RoboDK station: Colour sorting robot.rdk

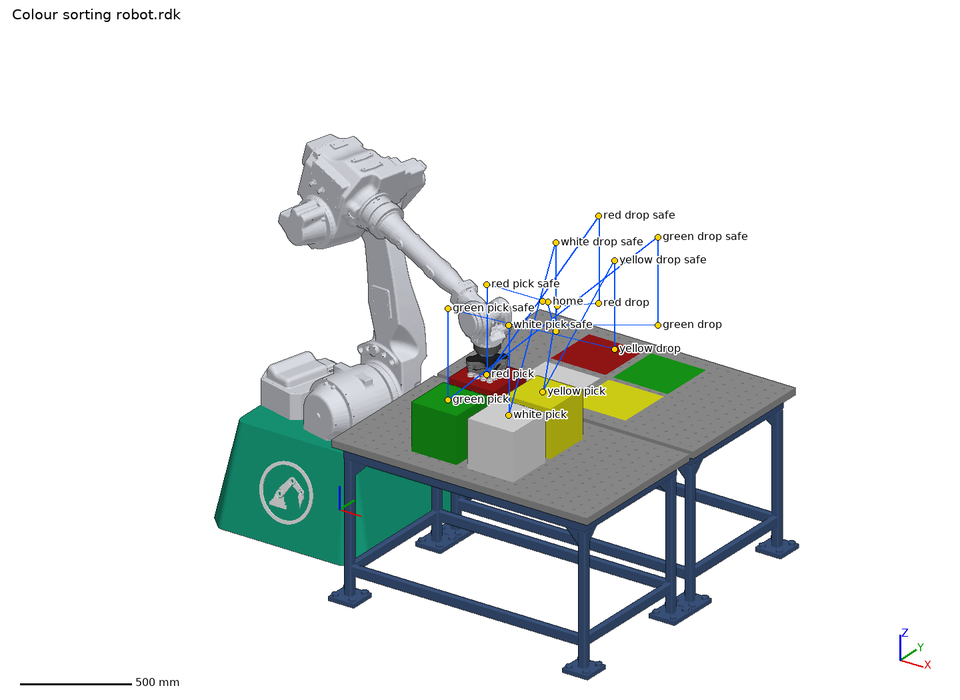
[picture v0: the station drawn from its stored meshes, robots at their saved joint values, targets as dots, program paths as lines]
Station nt colour sorting robot (saved by RoboDK 5.6.8). Poses are relative to the parent item; angles as X-Y-Z fixed-axis rotations.
  - frame Mitsubishi RV-35F Base at (0, 0, 0) mm
    - robot Mitsubishi RV-35F: 6 axes, payload 35 kg, reach 2050 mm, repeatability 0.07 mm
        modified DH rows (alpha deg, a mm, theta deg, d mm): 0, 0, 0, 600; -90, 150, -90, 0; 0, 900, -90, 0; -90, 150, 0, 990; 90, 0, 0, 0; -90, 0, 180, 175
        joint limits [-165, -80, -90, -360, -125, -450] to [165, 135, 171, 360, 125, 450]; home [0, 0, 90, 0, 0, 0]; saved at [-14.514, -7.868, 114.84, 0, 73.027, -14.514]
      - tool OnRobot VG10 Vacuum Gripper, TCP at (0, 0, 120.9) mm, size 145.4 x 145.4 x 118.3 mm
    - target home (Cartesian target) at (1140, 0, 1354.1) mm, rotated rx 180 ry 0 rz -180 deg; joints [0, 0, 90, 0, 90, 0] of Mitsubishi RV-35F
    - target red pick safe (Cartesian target) at (985, -255, 1500.1) mm, rotated rx 180 ry 0 rz -180 deg; joints [-14.514, -5.594, 86.759, 0, 98.836, -14.514] of Mitsubishi RV-35F
    - target red pick (Cartesian target) at (985, -255, 1050.1) mm, rotated rx 180 ry 0 rz -180 deg; joints [-14.514, -7.868, 114.84, 0, 73.027, -14.514] of Mitsubishi RV-35F
    - target red drop safe (Cartesian target) at (995, 605, 1500) mm, rotated rx 180 ry 0 rz -180 deg; joints [31.301, 3.727, 77.585, 0, 98.687, 31.301] of Mitsubishi RV-35F
    - target red drop (Cartesian target) at (995, 605, 1064) mm, rotated rx 180 ry 0 rz -180 deg; joints [31.301, 1.465, 105.177, 0, 73.358, 31.301] of Mitsubishi RV-35F
    - target yellow pick safe (Cartesian target) at (1370, -255, 1500.1) mm, rotated rx 180 ry 0 rz -180 deg; joints [-10.544, 19.818, 58.38, 0, 101.801, -10.544] of Mitsubishi RV-35F
    - target yellow pick (Cartesian target) at (1290, -255, 1050.1) mm, rotated rx 180 ry 0 rz -180 deg; joints [-11.182, 11.089, 95.402, 0, 73.509, -11.182] of Mitsubishi RV-35F
    - target yellow pick safe (Cartesian target) at (1290, -255, 1500) mm, rotated rx 180 ry 0 rz -180 deg; joints [-11.182, 13.953, 65.877, 0, 100.171, -11.182] of Mitsubishi RV-35F
    - target yellow drop safe (Cartesian target) at (1315, 270, 1500) mm, rotated rx 180 ry 0 rz -180 deg; joints [11.603, 15.946, 63.394, 0, 100.66, 11.603] of Mitsubishi RV-35F
    - target yellow drop (Cartesian target) at (1315, 270, 1060) mm, rotated rx 180 ry 0 rz -180 deg; joints [11.603, 12.747, 92.862, 0, 74.391, 11.603] of Mitsubishi RV-35F
    - target green pick safe (Cartesian target) at (985, -560, 1500) mm, rotated rx 180 ry 0 rz -180 deg; joints [-29.619, 1.694, 79.709, 0, 98.597, -29.619] of Mitsubishi RV-35F
    - target green pick (Cartesian target) at (985, -560, 1045) mm, rotated rx 180 ry 0 rz -180 deg; joints [-29.619, -0.352, 108.109, 0, 72.243, -29.619] of Mitsubishi RV-35F
    - target green pick safe (Cartesian target) at (985, -560, 1500) mm, rotated rx 180 ry 0 rz -180 deg; joints [-29.619, 1.694, 79.709, 0, 98.597, -29.619] of Mitsubishi RV-35F
    - target green drop safe (Cartesian target) at (1335, 580, 1500) mm, rotated rx 180 ry 0 rz -180 deg; joints [23.483, 24.904, 51.434, 0, 103.662, 23.483] of Mitsubishi RV-35F
    - target green drop (Cartesian target) at (1335, 580, 1060) mm, rotated rx 180 ry 0 rz -180 deg; joints [23.483, 20.031, 83.722, 0, 76.247, 23.483] of Mitsubishi RV-35F
    - target white pick safe (Cartesian target) at (1305, -540, 1500) mm, rotated rx 180 ry 0 rz -180 deg; joints [-22.479, 21.303, 56.401, 0, 102.296, -22.479] of Mitsubishi RV-35F
    - target white pick (Cartesian target) at (1305, -540, 1050) mm, rotated rx 180 ry 0 rz -180 deg; joints [-22.479, 17.288, 87.832, 0, 74.879, -22.479] of Mitsubishi RV-35F
    - target white drop safe (Cartesian target) at (995, 270, 1500) mm, rotated rx 180 ry 0 rz -180 deg; joints [15.182, -4.757, 85.998, 0, 98.759, 15.182] of Mitsubishi RV-35F
    - target white drop (Cartesian target) at (995, 270, 1060) mm, rotated rx 180 ry 0 rz -180 deg; joints [15.182, -7.076, 113.57, 0, 73.506, 15.182] of Mitsubishi RV-35F
  - object Table 1400x800x800mm at (840, -380, 800) mm, size 1420 x 820 x 800 mm, geometry from Table-1400x800x800mm (4).sld
  - object Pedestal H500mm (Type 2) at (0, 0, 0) mm, size 844.5 x 933.7 x 500 mm, geometry from Pedestal-H500mm-Type-2.sld
  - object Table 1400x800x800mm at (840, 450, 800) mm, size 1420 x 820 x 800 mm, geometry from Table-1400x800x800mm (4).sld
  - object Square at (990, 600, 810) mm, size 300 x 300 x 0 mm, geometry from Square.sld
  - object Square at (990, 260, 810) mm, size 300 x 300 x 0 mm, geometry from Square.sld
  - object Square at (1330, 600, 810) mm, size 300 x 300 x 0 mm, geometry from Square.sld
  - object Square at (1330, 270, 810) mm, size 300 x 300 x 0 mm, geometry from Square.sld
  - program attach (1 instructions, listed below)
  - program detach (1 instructions, listed below)
  - program reset (1 instructions, listed below)
  - program main (29 instructions, listed below)
  - object cube2 at (860, 0, 800) mm, size 250 x 250 x 250 mm, geometry from Cube-500mm.sld
  - object cube4 at (1170, -380, 800) mm, size 250 x 250 x 250 mm, geometry from Cube-500mm.sld
  - object cube1 at (860, -670, 794.9) mm, size 250 x 250 x 250 mm, geometry from Cube-500mm.sld
  - object cube3 at (1170, -670, 799.9) mm, size 250 x 250 x 250 mm, geometry from Cube-500mm.sld
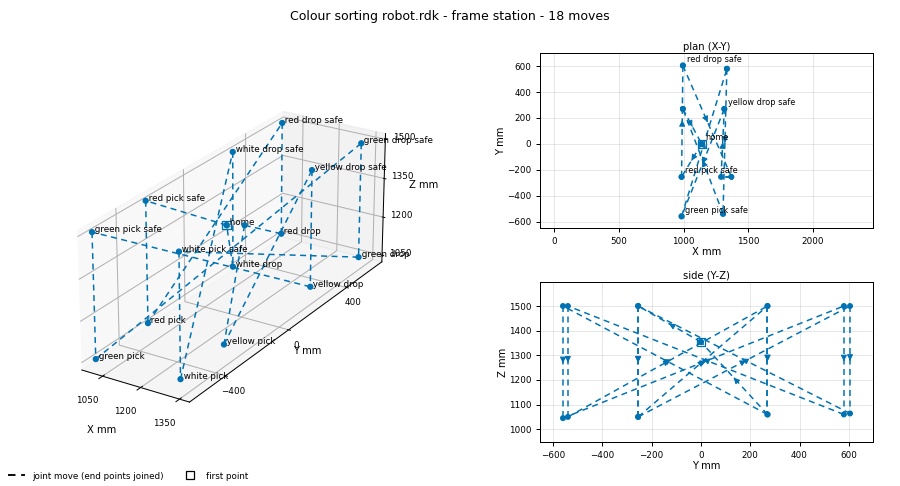
[picture p0: tool path of Colour sorting robot.rdk in frame station, 18 of 18 moves have a stored position in this frame; points joined in program order, loops and branches not executed]

--- program attach (robot Mitsubishi RV-35F) ---
  Attach to OnRobot VG10 Vacuum Gripper

--- program detach (robot Mitsubishi RV-35F) ---
  Detach from OnRobot VG10 Vacuum Gripper

--- program reset (robot Mitsubishi RV-35F) ---
  Replace objects

--- program main (robot Mitsubishi RV-35F) ---
  Set Ref.: Mitsubishi RV-35F Base
  Set Tool: OnRobot VG10 Vacuum Gripper
  MoveJ (home)
  MoveJ (red pick safe)
  MoveJ (red pick)
  Call attach
  MoveJ (red drop safe)
  MoveJ (red drop)
  Call detach
  MoveJ (yellow pick safe)
  MoveJ (yellow pick)
  Call attach
  MoveJ (yellow drop safe)
  MoveJ (yellow drop)
  Call detach
  MoveJ (green pick safe)
  MoveJ (green pick)
  Call attach
  MoveJ (green drop safe)
  MoveJ (green drop)
  Call detach
  MoveJ (white pick safe)
  MoveJ (white pick)
  Call attach
  MoveJ (white drop safe)
  MoveJ (white drop)
  Call detach
  MoveJ (home)
  Call reset
